// TIA Portal V19 export
TYPE "LEXCHANGETRAY_typeConstraintRollerEm_xPositionAxis_moduleInterface"
// stored: Access Published
   STRUCT
      axisControlModuleInterface : "LBC_typeAxisSimpleControlInterface_1";
      xPosConfigeration : "LEXCHANGETRAY_typeConstraintRollerEm_xPositionAxis_configuration";
      xPosmonitor { S7_SetPoint := 'True'} : "LEXCHANGETRAY_typeConstraintRollerEm_xPositionAxis_monitor";
   END_STRUCT;
END_TYPE
